# EPICS IOC start-up script: examples/test/PSI/epp2008.iocsh
#- mXsXXX naming
require ecmccfg, "NAMING=mXsXXX"

#- add slaves
${SCRIPTEXEC} ${ecmccfg_DIR}addSlave.cmd, "HW_DESC=EPP2008, SLAVE_ID=3"
